METHOD raiseError
VAR_INPUT
	bSetError : BOOL;
END_VAR
CASE iErrorId OF
	C234_FEEDMANAGER_FAILED_TO_FIND_FALLING_EDGE_OF_C_OR_D_FEED_EYE: 
		formatError('Failed to find falling edge of C or D feed eye', 'Turn Autofeed on and retry');
	C234_FEEDMANAGER_DOWNSTREAM_ERROR: 
		formatError('Downstream error', 'Reset machine');
	C234_FEEDMANAGER_FAILED_TO_FIND_OUTFEED_END_EYE: 
		formatError('Failed to find the outfeed-end eye', 'Turn Autofeed on and retry');
	C234_FEEDMANAGER_C_AND_D_FEED_EYES_MUST_BE_CLEAR: 
		formatError('C and D feed eyes must be clear', 'Turn Autofeed on and retry');
	C234_FEEDMANAGER_FEEDIN_FAILED_TO_FIND_STOP_EYE_1_RISING_EDGE_OR_INFEED_EYE: 
		formatError('Failed to find door-stop eye 1 rising edge or infeed eye falling edge during feed-in sequence', 'Turn Autofeed on and retry');
	C234_FEEDMANAGER_INIT_FAILED_TO_FIND_STOP_EYE_1_RISING_EDGE_OR_INFEED_EYE: 
		formatError('Failed to find door-stop eye 1 rising edge or infeed eye falling edge during init sequence', 'Turn Autofeed on and retry');
	C234_FEEDMANAGER_FAILED_TO_FIND_STOP_EYE_1_RISING_EDGE: 
		formatError('Failed to find door-stop eye 1 rising edge', 'Turn Autofeed on and retry');
	C234_FEEDMANAGER_FAILED_TO_FIND_STOP_EYE_3_RISING_EDGE: 
		formatError('Failed to find door-stop eye 3 rising edge', 'Turn Autofeed on and retry');		
	C234_FEEDMANAGER_FAILED_TO_FIND_IN_MACHINE_EYE: 
		formatError('Failed to find in-machine eye', 'Turn Autofeed on and retry');
	C234_FEEDMANAGER_FAILED_TO_FIND_FENCE_EYE_RISING_EDGE: 
		formatError('Failed to find fence eye rising edge', 'Turn Autofeed on and retry');
END_CASE
SUPER^.raiseError(bSetError);
END_METHOD

(* base implementation to record state calling history. 
 	Derrived FB's should override this method to replace the machine' specific type of eState *)
	
METHOD recordStateCallHistory
VAR_INPUT
	iState				: INT;
	iSubState			: INT;
END_VAR
VAR
	sCurTaskCycle 		: STRING;
    eState       		: E_234FeedManager_States; // todo: replace with the derrived STRUCT type (ie, E_HeadManager_States)
    eSubState			: E_SubState;
END_VAR
// DO NOT CHANGE BELOW!!!
// This was auto-generated by a Kval's UML tool.

sCurTaskCycle := TO_STRING(mainStateCallingData[iState, iSubState].nCycleIdFirstCall);
eState := iState;
eSubState := iSubState;

// Enter the state name into array
mainStateCallHistory[iStateCallHistoryIndex].sTaskCycle := sCurTaskCycle;
mainStateCallHistory[iStateCallHistoryIndex].sStateId := TO_STRING(iState);
mainStateCallHistory[iStateCallHistoryIndex].sStateDesc := TO_STRING(eState);
mainStateCallHistory[iStateCallHistoryIndex].sSubStateId := TO_STRING(iSubState);
mainStateCallHistory[iStateCallHistoryIndex].sSubStateDesc := TO_STRING(eSubState);

iStateCallHistoryIndex := iStateCallHistoryIndex + 1;
IF iStateCallHistoryIndex = MAX_STATE_CALL_HISTORY THEN
	iStateCallHistoryIndex := 0;
END_IF

// mark next index to record state call history
mainStateCallHistory[iStateCallHistoryIndex].sTaskCycle := '--';
mainStateCallHistory[iStateCallHistoryIndex].sStateId := '--';
mainStateCallHistory[iStateCallHistoryIndex].sStateDesc := '--';
mainStateCallHistory[iStateCallHistoryIndex].sSubStateId := '--';
mainStateCallHistory[iStateCallHistoryIndex].sSubStateDesc := '--';
END_METHOD

METHOD resetFeedinDoorsCount
VAR_INPUT
END_VAR
iFeedoutDoorsCount := 0;
END_METHOD

(* Any trigger that caused state transition (ie, cmd_bHome, cmd_bStartSequence, etc..) that
 	needs to be reset should go in here.
	 
	NOTE: The derived function block of KvalStateMachineBase_UmlSC should override/extend this method. *)
METHOD resetTriggers
SUPER ^.resetTriggers();
//TODO: reset all triggers (ie, cmd_bHome, cmd_bPark, etc...) here...
END_METHOD

METHOD setDisableFeedoutSideA
VAR_INPUT
	bDisableFeedoutSideA : BOOL;
END_VAR
IF config_bNoHardwareTestMode THEN
	di_DisableFeedoutSideA := bDisableFeedoutSideA;
END_IF
END_METHOD

METHOD setDisableFeedoutSideB
VAR_INPUT
	bDisableFeedoutSideB : BOOL;
END_VAR
IF config_bNoHardwareTestMode THEN
	di_DisableFeedoutSideB := bDisableFeedoutSideB;
END_IF
END_METHOD

METHOD setDoorDataAck
VAR_INPUT
	bDoorDataAck : BOOL;
END_VAR
do_DoorDataAck := bDoorDataAck;
END_METHOD

METHOD setReadyToFeedoutSideA
VAR_INPUT
	bReadyToFeedoutSideA : BOOL;
END_VAR
do_ReadyToFeedoutSideA := bReadyToFeedoutSideA;
END_METHOD

METHOD setReadyToFeedoutSideB
VAR_INPUT
	bReadyToFeedoutSideB : BOOL;
END_VAR
do_ReadyToFeedoutSideB := bReadyToFeedoutSideB;
END_METHOD

METHOD setRotationRequired
VAR_INPUT
END_VAR
bRotateRequired := 
	NOT bInitRunning AND 				 
	config_bCanRotate AND 
	(pstDoorTrack^.DoorRotateRequired XOR pstDoorTrack^.DoorWasRotated)	
;
END_METHOD

METHOD setTableEmptyStatus
VAR_INPUT
	bEmpty : BOOL;
END_VAR
SUPER^.setTableEmptyStatus(bEmpty);
pbTableIsEmpty^ := bEmpty;
bDoorInMachine := NOT bEmpty;
pbDoorInMachine^ := bDoorInMachine;
END_METHOD

(* Each transition has either or both a trigger (ie, cmd_bHome, cmd_bStartSequence, etc..)
	and a guard condition (i.e., bHeadReady AND bTableReady).
	This method updates all the state transitions.
	 
	NOTE: The derived function block of KvalStateMachineBase_UmlSC MUST override/extend this method. *)
METHOD updateStateTransitions
END_METHOD

END_FUNCTION_BLOCK

(* stored: Version 1.1.0.1, ProductVersion 3.1.4024.13
   POU SM_234FeedManager: Id {4e540ff9-af90-451c-8463-b311a5dc8289}, SpecialFunc None
   Folder uml: Id {ffa918be-ea15-4341-940c-4bb585c193dc}
   Method blinkReadyToFeedoutSideA: Id {fa00e0e7-7172-4d21-92a7-8fabebeb8502}
   Method blinkReadyToFeedoutSideB: Id {d1f94fcd-d39d-40e8-845b-7630cca7d3fb}
   Method destinationDigitalInputsToDestinationIndex: Id {458713c3-c9b7-438f-adba-a06555fd4e47}
   Method doState: Id {44cf212b-2e1e-472c-87eb-5d80e83b9bbd}
   Method doState_UmlSC: Id {389a986f-65e9-4078-891d-a48267681975}
   Method getStateDescription: Id {15b7f27f-d611-4c41-a1b8-0d471853890a}
   Method initialize: Id {1a82f989-738b-45ac-bc9f-52d263f74b91}
   Method isTableEmpty: Id {17b4c1b7-78a7-4f06-9d3c-e2ea5d004a76}
   Method postProcess: Id {6a82d0bf-ecbb-4165-b4e2-33a45c0d701e}
   Method preProcess: Id {6725ecf3-ae81-46de-9298-467dcfdee35f}
   Method raiseError: Id {251b2b3f-3bca-444d-9b5d-fa3b9857a089}
   Method recordStateCallHistory: Id {e598d84d-220c-4eb4-acca-e2dcd76e780d}
   Method resetFeedinDoorsCount: Id {ed189374-0ced-45e5-a713-66f74f7b7913}
   Method resetTriggers: Id {1283b628-9c94-4814-a913-94fb25243562}
   Method setDisableFeedoutSideA: Id {ce90d296-0aa9-4def-8832-ba89a3be0ab6}
   Method setDisableFeedoutSideB: Id {de919d2b-770a-4d3b-a44a-5830c967dfc3}
   Method setDoorDataAck: Id {e6455d20-fc7b-434e-b056-7418125bad51}
   Method setReadyToFeedoutSideA: Id {1cc6400c-552b-4615-adf7-fa88e76071f1}
   Method setReadyToFeedoutSideB: Id {d2ee0db6-5c76-4a69-be70-846fd392b829}
   Method setRotationRequired: Id {a18d8cc1-b479-4d2a-8082-68df5d753eec}
   Method setTableEmptyStatus: Id {8d8696f2-d89e-45b6-a8d0-df7af61454ce}
   Method updateStateTransitions: Id {25b19d1a-2df7-48e9-ac4a-966c84d52276} *)
